(* PLC project LorochCxPlc_1, Beckhoff Automation GmbH TwinCAT PLC Control 3.5.13.20 *)
(* stored: creationDateTime 2020-11-20T11:41:12.3628683, modificationDateTime 2020-11-20T11:41:12.3628683 *)

{attribute 'pack_mode' := '1'}
TYPE ST_MachSpecificRaw :
	STRUCT
				(* checksum *)
					Raw100			:	LREAL;
				(* base *)
					Raw1000			:	INT;
					Raw1001			:	STRING;
					Raw1002			:	INT;
					Raw1003			:	STRING;
					Raw1004			:	ARRAY[0..3] OF REAL;
					Raw2010			:	ARRAY[0..7] OF BOOL;
					Raw2020			:	ARRAY[0..1] OF BOOL;
					Raw2021			:	BOOL;
					Raw2022			:	ARRAY[0..5] OF UINT;
					Raw2023			:	ARRAY[0..2] OF BOOL;
					Raw2024			:	ARRAY[0..2] OF REAL;
					Raw2025			:	ARRAY[0..1] OF BOOL;
					Raw2030			:	ARRAY[0..2] OF BOOL;
				(* UI visu *)
					Raw2040			:	ARRAY[0..7] OF BOOL;
					Raw2050			:	INT;
				(* ui config *)
				(* peripheral basic *)
				(* axis *)
				(* x axis *)
					Raw3000			:	BOOL;
					Raw3001			:	ARRAY[0..1] OF INT;
					Raw3002 		:	ARRAY[0..11] OF REAL;
					Raw3003 		:	ARRAY[0..1] OF LREAL;
				(* y axis *)
					Raw3100			:	BOOL;
					Raw3101			:	ARRAY[0..1] OF INT;
					Raw3102 		:	ARRAY[0..11] OF REAL;
					Raw3103 		:	ARRAY[0..3] OF REAL;
				(* z axis *)
					Raw3200			:	BOOL;
					Raw3201			:	ARRAY[0..1] OF INT;
					Raw3202 		:	ARRAY[0..11] OF REAL;
					Raw3203 		:	ARRAY[0..3] OF REAL;
				(* axis position *)
					Raw3300			:	ARRAY[0..1] OF REAL;
				(* coolant/filter *)
				(* chiller *)
					Raw4000			:	BOOL;
					Raw4001			:	REAL;
					Raw4002 		:	BOOL;
				(* filter *)
					Raw4100			:	BOOL;
					Raw4101			:	REAL;
					Raw4102 		:	BOOL;
				(* return feed pump *)
					Raw4200			:	BOOL;
					Raw4201			:	REAL;
					Raw4202 		:	BOOL;
				(* coolant pump *)
					Raw4300			:	BOOL;
					Raw4301			:	REAL;
					Raw4302 		:	BOOL;
				(* cartridge counter *)
					Raw4400			:	ARRAY[0..2] OF UINT;
				(* Extraction *)
					Raw5000			:	BOOL;
					Raw5001			:	REAL;
				(* grinding head *)
					Raw6000			:	INT;
				(* grinding wheel *)
				(* cbn *)
					Raw7000			:	BOOL;
					Raw7001			:	STRING[3];
					Raw7002 		:	ARRAY[0..2] OF REAL;
				(* dia - carbide *)
					Raw7100			:	BOOL;
					Raw7101			:	STRING[3];
					Raw7102 		:	ARRAY[0..2] OF REAL;
				(* dia - cermet *)
					Raw7200			:	BOOL;
					Raw7201			:	STRING[3];
					Raw7202 		:	ARRAY[0..2] OF REAL;
				(* dressing *)
					Raw7300			:	BOOL;
					Raw7301			:	STRING[3];
					Raw7302 		:	ARRAY[0..2] OF REAL;
				(* lubrication *)
					Raw8000			:	ARRAY[0..1] OF UINT;
				(* peripheral basic *)
				(* peripheral optional *)
				(* chip breaker *)
					Raw9000			:	BOOL;
					Raw9001			:	INT;
					Raw9002			:	ARRAY[0..1] OF UINT;
					Raw9003			:	ARRAY[0..3] OF REAL;
				(* fire extinguisher *)
					Raw10000		:	ARRAY[0..1] OF BOOL;
				(* flange handler *)
					Raw11000		:	INT;
					Raw11001		:	BOOL;
				(* res - not longer used for flange handler *)
					Raw11002		:	ARRAY[0..11] OF REAL;
				(* light barrier *)
					Raw12000		:	BOOL;
					Raw12001		:	UINT;
					Raw12002		:	BOOL;
					Raw12003		:	ARRAY[0..1] OF REAL;
				(* positioning sensor *)
					Raw13000		:	ARRAY[0..3] OF BOOL;
				(* loader*)
					Raw14000		:	BOOL;
					Raw14001		:	ARRAY[0..1] OF REAL;
					Raw14002		:	UINT;
				(* saw blade clamping *)
					Raw15000		:	ARRAY[0..1] OF BOOL;
				(* saw blade handler *)
					Raw16000		:	BOOL;
					Raw16001		:	INT;
					Raw16002		:	ARRAY[0..4] OF DINT;
				(* support bracket *)
					Raw17000		:	BOOL;
					Raw17001		:	INT;
					Raw17002		:	ARRAY[0..2] OF BOOL;
				(* peripheral optional *)
				(* peripheral basic *)
				(* safety controller *)
					Raw18000		:	INT;
				(* peripheral basic *)
				(* new opmode *)
					Raw19000		:	ARRAY[0..7] OF BOOL;
				(* new toothshape *)
					Raw19001		:	ARRAY[0..7] OF BOOL;
				(* new chipbreaker *)
					Raw19200		:	ARRAY[0..1] OF REAL;
					Raw19201		:	ARRAY[0..1] OF REAL;
				(* touch man handwheel mode *)
					Raw19300		:	INT;
				(* new StoringOptions *)
					Raw19310		:	ARRAY[0..3] OF BOOL;
				(* new ProcessingOptions *)
					Raw19320		:	ARRAY[0..1] OF INT;
				(* new FRed *)
					Raw19330		:	INT;
					Raw19331		:	INT;
				(* support bracket message delay *)
					Raw19340		:	REAL;
				(* loader *)
					Raw19400		:	ARRAY[0..1] OF INT;
					Raw19410		:	ARRAY[0..5] OF REAL;
				(* hydraulics *)
					Raw19420		:	BOOL;
				(* voltage monitoring *)
					Raw19430		:	BOOL;
				(* lubrication circuit 2 *)
					Raw19440		:	BOOL;
					Raw19441		:	ARRAY[0..1] OF UINT;
				(* ethercat *)
					Raw19450		:	UINT;
				(* homing pos *)
					Raw19460		:	REAL;
				(* New Loader Arbor *)
					Raw19500		:	UINT;	(* ArborNumber *)
					Raw19510		:	UINT;	(* ArborNumberSource	*)
				(* New CachedStacks *)
					Raw19550		:	UINT;
					Raw19600		:	UINT;(* Neu *)
				(* Infeed Correction chamfering *)
					Raw19650		:	ARRAY[0..1] OF BOOL;
					Raw19651		:	ARRAY[0..5] OF REAL;
				(* axis options *)
					Raw19655		:	ARRAY[0..4] OF BOOL;
				(* UI visu *)
					Raw19700		:	BOOL;
				(* LightBarrier PositionOffset *)
					Raw19710		:	REAL;
				(* positioning sensor*)
					Raw19800		:	BOOL;
					Raw19801		:	INT;
				(* SawBladeMeasureAuto *)
					Raw19810		:	BOOL;
				(* OperatingModeTouchOption *)
					Raw19811		:	BOOL;
				(* CoolantSystem *)
					Raw19814		:	INT;
				(* FeedRateCorrection *)
					Raw19815		:	REAL;
				(* grinding head no swivel at process end *)
					Raw19820		:	BOOL;
				(* remote monitoring *)
					Raw19825		:	ARRAY[0..2] OF BOOL;
					Raw19830		:	ARRAY[0..1] OF REAL;
					Raw19831		:	REAL;
				(* Safety Circuit Option : With/Without Enabling Switches *)
					Raw19833		:	INT;
				(* Chip Breaker Motion Type *)
					Raw19835		:	 INT;	(* Stepper , Pneumatic *)
					Raw19839		:	REAL;	(* Reference position of the stepper Motor *)
					Raw19840		:	ARRAY[0..3] OF REAL; (* New for ChipBreaker GW Width and Diameter *)
				(* info -> Raw11002 = res *)
				(* grinding wheel model *)
					Raw19842		:	INT;
				(* limit switch z axis *)
					Raw19843		:	BOOL;
				(* lubrication *)
					Raw19844		:	ARRAY[0..1] OF BOOL;
				(* pneumatics *)
					Raw19845		:	BOOL;
				(* temperature monitoring *)
					Raw19846		:	BOOL;
				(* limit switch normally open / pressure switch - coolant ystem *)
					Raw19847		:	ARRAY[0..4] OF BOOL;
				(* limit switch normally open - extraction *)
					Raw19848		:	BOOL;

				(* Chip Breaker Edge Distance *)
					Raw19850		:	INT;
					Raw19851		:	REAL;
					Raw19852		:	BOOL;
					Raw19853		:	REAL;
					Raw19854		:	BOOL;
				(* Remote monitoring fire extinguisher ext warning *)
					Raw19856		:	BOOL;
				(* Grinding Wheel Cover *)
					Raw19860		:	INT;
				(* Chamfer No of Touch *)
					Raw19865		:	ARRAY[0..1] OF UINT;
				(* chamfer touch pos *)
					Raw19866		:	ARRAY[0..1] OF BOOL;
				(* History File *)
					(* writing Conditions *)
					Raw19868		:	ARRAY [0..1] OF BOOL;
				(* History File Buffering *)
					Raw19869		:	UINT;
					(* Extraction Running Monitoring *)
					Raw19870		:	BOOL;
				(* FRed Chamfering InFeed *)
					Raw19880		:	ARRAY[0..5] OF BOOL;
					Raw19881		:	ARRAY[0..5] OF REAL;
					Raw19885		:	BOOL;
					Raw19886		:	LREAL;
					Raw19887		:	BOOL;
				(*  FRed ExpandedOrders *)
					Raw19888		:	UINT;
				(* ThinKerfCuttingInsert *)
					Raw19890		:	ARRAY[0..5] OF BOOL;	(*ARRAY[0..5] OF BOOL;*)
					Raw19892		:	ARRAY[0..3] OF UINT;
					Raw19894		:	ARRAY[0..3] OF INT;
					Raw19896		:	ARRAY[0..3] OF INT;
					Raw19898		:	ARRAY[0..14,0..1] OF REAL;
				(*TKT Light Barrier*)
					Raw19900		:	BOOL;
					Raw19902		:	REAL;
					(* ThinKerfCuttingInsert *)
					Raw19905		:	ARRAY [0..1] OF BOOL;
					Raw19907        :	ARRAY [0..3] OF BOOL;
					(* SelectMultipleOrders SelectMultipleStacks *)
					Raw19908		:	ARRAY[0..1] OF BOOL;
					
				(* HardItem *)
					(* base *)
						(* twincat version *)
						Raw19910		:	INT;
						(* sawblade dimension limits *)
						Raw19912		:	ARRAY[0..7] OF REAL;
						(* working angle *)
						Raw19914		:	REAL;
					(* uiconfiguration *)
						(* storing options *)
						Raw19916		:	BOOL; 
						(* positioning mode *)
						Raw19918		:	ARRAY[0..2] OF BOOL;
						(* chamfering *)
						Raw19920		:	BOOL;
						(* chamfering - chamfer width default, Main cutting edge default *)
						Raw19922		:	ARRAY[0..1] OF BOOL;
						(* chamfering - protection chamfer *)
						Raw19924		:	ARRAY[0..1] OF REAL;
						(* chamfering - protection chamfer 2 *)
						Raw19926		:	ARRAY[0..1] OF REAL;
						(* carbide tip seat *)
						Raw19928		:	BOOL;
						(* relief grinding *)
						Raw19930		:	BOOL;
						(* repairing tooth *)
						Raw19932		:	BOOL;
						(* tooth construction - saw blade category *)
						Raw19934		:	ARRAY[0..1] OF BOOL;
						(* tooth construction - saw blade geometry *)
						Raw19936		:	ARRAY[0..8] OF BOOL;
						(* tooth construction - clearance surface back *)
						Raw19938		:	ARRAY[0..1] OF BOOL;
					(* peripheral basic *)
						(* axis *)
						(* axis - v axis *)
						Raw19940		:	BOOL;
						Raw19942		:	ARRAY[0..1] OF INT;
						Raw19944 		:	ARRAY[0..11] OF LREAL;
						Raw19946 		:	ARRAY[0..1] OF REAL;
						Raw19948		:	ARRAY[0..4,0..1] OF REAL;
						(* axis - w axis *)
						Raw19950		:	BOOL;
						Raw19952		:	ARRAY[0..1] OF INT;
						Raw19954 		:	ARRAY[0..11] OF LREAL;
						Raw19956 		:	ARRAY[0..1] OF REAL;
						Raw19958		:	ARRAY[0..4,0..1] OF REAL;
						(* lubrication - circuit 1 *)
						Raw19960		:	BOOL;
						Raw19962		:	INT;
						Raw19964 		:	ARRAY[0..1] OF UINT;
						Raw19966 		:	REAL;
						(* lubrication - circuit 2 *)
						Raw19968		:	BOOL;
						Raw19970		:	INT;
						Raw19972 		:	ARRAY[0..1] OF UINT;
						Raw19974 		:	REAL;
						(* grinding wheel *)
						(* grinding wheel - lead angle default *)
						Raw19976		:	REAL;
						(* grinding wheel - cermet *)
						Raw19978		:	BOOL;
						Raw19980 		:	ARRAY[0..1] OF INT;
						Raw19982 		:	ARRAY[0..2] OF REAL;
						(* grinding wheel - carbide *)
						Raw19984		:	BOOL;
						Raw19986 		:	ARRAY[0..1] OF INT;
						Raw19988 		:	ARRAY[0..2] OF REAL;
						(* grinding wheel - steel *)
						Raw19990		:	BOOL;
						Raw19992 		:	ARRAY[0..1] OF INT;
						Raw19994 		:	ARRAY[0..2] OF REAL;
					(* peripheral optional *)
						(* remote monitoring *)
						(* remote monitoring - to external *)
						Raw19996 		:	ARRAY[0..7] OF INT;
						(* remote monitoring - from external *)
						Raw19998 		:	ARRAY[0..7] OF INT;
						(* io link *)
						Raw20000		:	UINT;
	END_STRUCT
END_TYPE
